{attribute 'qualified_only'}
VAR_GLOBAL

END_VAR

VAR_GLOBAL CONSTANT
    axisNum :   UINT:=10;
END_VAR

(* stored: Version 1.1.0.1, ProductVersion 3.1.4024.2
   GVL GVL_APP: Id {8fe9690c-7907-432e-bedb-6fc99b5ce255} *)
